{library PUBLIC}
TYPE INFO_FUNCTION_NUMBER :(
	INFO_FUNCTION_RPC_STATUS:=1,				(* Get RPC call status *)
	INFO_FUNCTION_SYSTEM_STATUS:=2				(* Get system status *)
);
END_TYPE

(* stored: Version 1.1.0.1, ProductVersion 3.1.4022.12
   EnumerationTextList INFO_FUNCTION_NUMBER: Id {d6b9c090-dd70-4dcc-96ce-b43b2e08dffe} *)
